FUNCTION_BLOCK FB_Mode
VAR_INPUT
	iManualMode:				BOOL; //manual button
	iAutoMode:					BOOL; //auto button
	iStartAutoCycle:			BOOL; //start auto cycle button
	iStopAutoCycle:				BOOL; //stop Auto cycle
	iStopEOC:					BOOL; //stop end of cycle
	iSemiAutoMode:				BOOL; //semi auto button
	iContCycle:					BOOL; //continuous cycle mode
	iSingleCycle:				BOOL; //single cycle mode
	iHome:						BOOL;  //station is at HOME
	iFault:						BOOL;
	iDryCycleMode:				BOOL; //station in dry cycle mode

	iIsStationSelected: BOOL; //is the current station selected?
	
	iLocalRemoteEnable: BOOL; //TRUE if the local station is in remote mode

	iRemoteData:typeRemote; //data from remote source
	
	iStartAutoCycleDelay:TIME:=T#2S; //delay time to start auto cycle
	iFirstScan:BOOL:=TRUE; //first scan logic for seting inital mode
	iStopCycleTimeout:TIME:=T#120S; //time to stop auto cycle if home not reached in (t). Set to 110% of expected station cycle time
	//isStationLocked:				BOOL;
END_VAR
	
	
VAR
	tAutoCycleStop: BOOL;
	timDelayRemoteOn: ton;
	ModeColourConv: FB_ModeStateToColour;
	timDelayAutoCycleStart: TON;
	timSEOCtimeout: TON;
	tUseOtherStation: BOOL;
	tResetSEOC: BOOL;
END_VAR

VAR_OUTPUT
END_VAR

VAR_IN_OUT
	stationState:typeStationMode;
	lockedModes:typeStationLockModes;
END_VAR
//theme:LYwABmhF6lY
VAR // added by the converter: edge detectors and wires of the graphical bodies
    _rt1, _rt2, _rt3, _rt4, _rt5, _rt6, _rt7, _rt8, _rt9, _rt10, _rt11, _rt12, _rt13, _rt14, _rt15, _rt16, _rt17, _rt18 : R_TRIG;
    _w1, _w2, _w3 : BOOL;
END_VAR

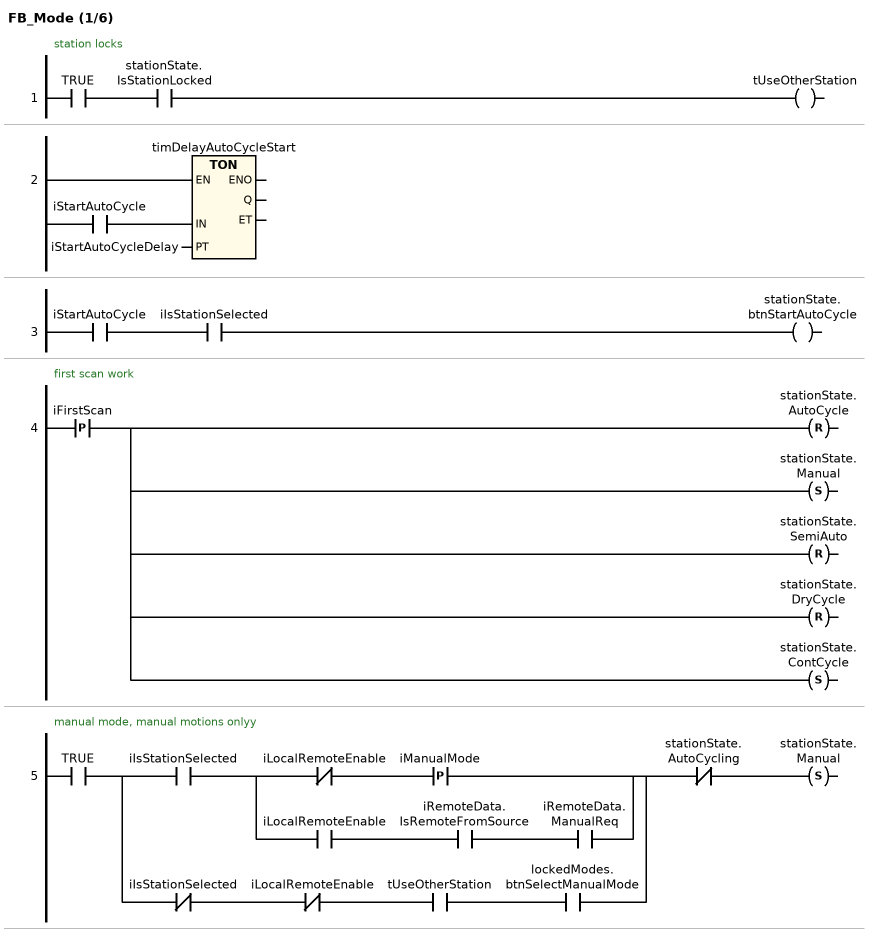
// NETWORK 1
// station locks
tUseOtherStation := TRUE AND stationState.IsStationLocked;

// NETWORK 2
timDelayAutoCycleStart(IN := iStartAutoCycle, PT := iStartAutoCycleDelay); // TON

// NETWORK 3
stationState.btnStartAutoCycle := iStartAutoCycle AND iIsStationSelected;

// NETWORK 4
// first scan work
_rt1(CLK := iFirstScan);
stationState.AutoCycle R= _rt1.Q;
stationState.Manual S= _rt1.Q;
stationState.SemiAuto R= _rt1.Q;
stationState.DryCycle R= _rt1.Q;
stationState.ContCycle S= _rt1.Q;

// NETWORK 5
// manual mode, manual motions onlyy
_rt2(CLK := iManualMode);
stationState.Manual S= TRUE AND (iIsStationSelected AND (NOT iLocalRemoteEnable AND _rt2.Q OR iLocalRemoteEnable AND iRemoteData.IsRemoteFromSource AND iRemoteData.ManualReq) OR NOT iIsStationSelected AND NOT iLocalRemoteEnable AND tUseOtherStation AND lockedModes.btnSelectManualMode) AND NOT stationState.AutoCycling;

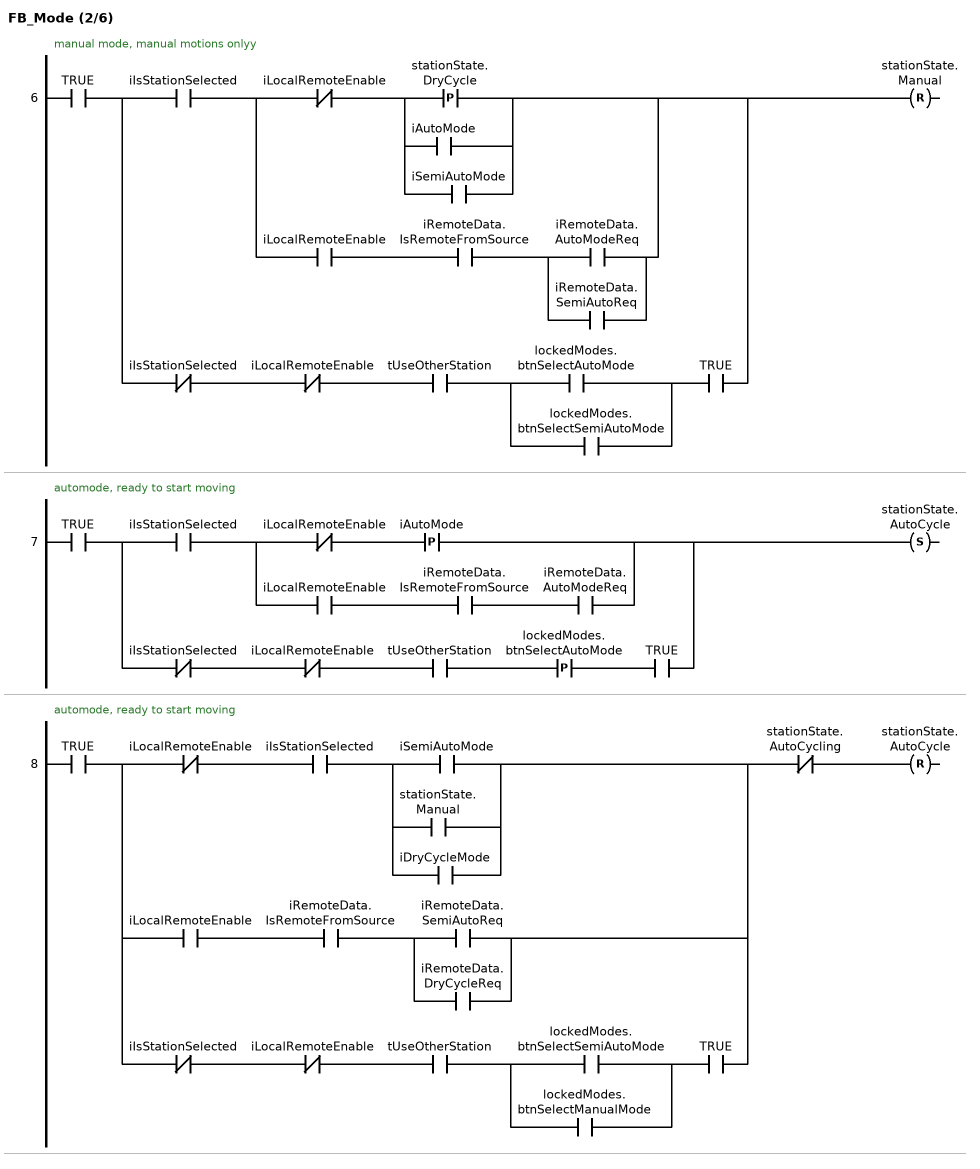
// NETWORK 6
// manual mode, manual motions onlyy
_rt3(CLK := stationState.DryCycle);
stationState.Manual R= TRUE AND (iIsStationSelected AND (NOT iLocalRemoteEnable AND (_rt3.Q OR iAutoMode OR iSemiAutoMode) OR iLocalRemoteEnable AND iRemoteData.IsRemoteFromSource AND (iRemoteData.AutoModeReq OR iRemoteData.SemiAutoReq)) OR NOT iIsStationSelected AND NOT iLocalRemoteEnable AND tUseOtherStation AND (lockedModes.btnSelectAutoMode OR lockedModes.btnSelectSemiAutoMode) AND TRUE);

// NETWORK 7
// automode, ready to start moving
_rt4(CLK := iAutoMode);
_rt5(CLK := lockedModes.btnSelectAutoMode);
stationState.AutoCycle S= TRUE AND (iIsStationSelected AND (NOT iLocalRemoteEnable AND _rt4.Q OR iLocalRemoteEnable AND iRemoteData.IsRemoteFromSource AND iRemoteData.AutoModeReq) OR NOT iIsStationSelected AND NOT iLocalRemoteEnable AND tUseOtherStation AND _rt5.Q AND TRUE);

// NETWORK 8
// automode, ready to start moving
stationState.AutoCycle R= TRUE AND (NOT iLocalRemoteEnable AND iIsStationSelected AND (iSemiAutoMode OR stationState.Manual OR iDryCycleMode) OR iLocalRemoteEnable AND iRemoteData.IsRemoteFromSource AND (iRemoteData.SemiAutoReq OR iRemoteData.DryCycleReq) OR NOT iIsStationSelected AND NOT iLocalRemoteEnable AND tUseOtherStation AND (lockedModes.btnSelectSemiAutoMode OR lockedModes.btnSelectManualMode) AND TRUE) AND NOT stationState.AutoCycling;

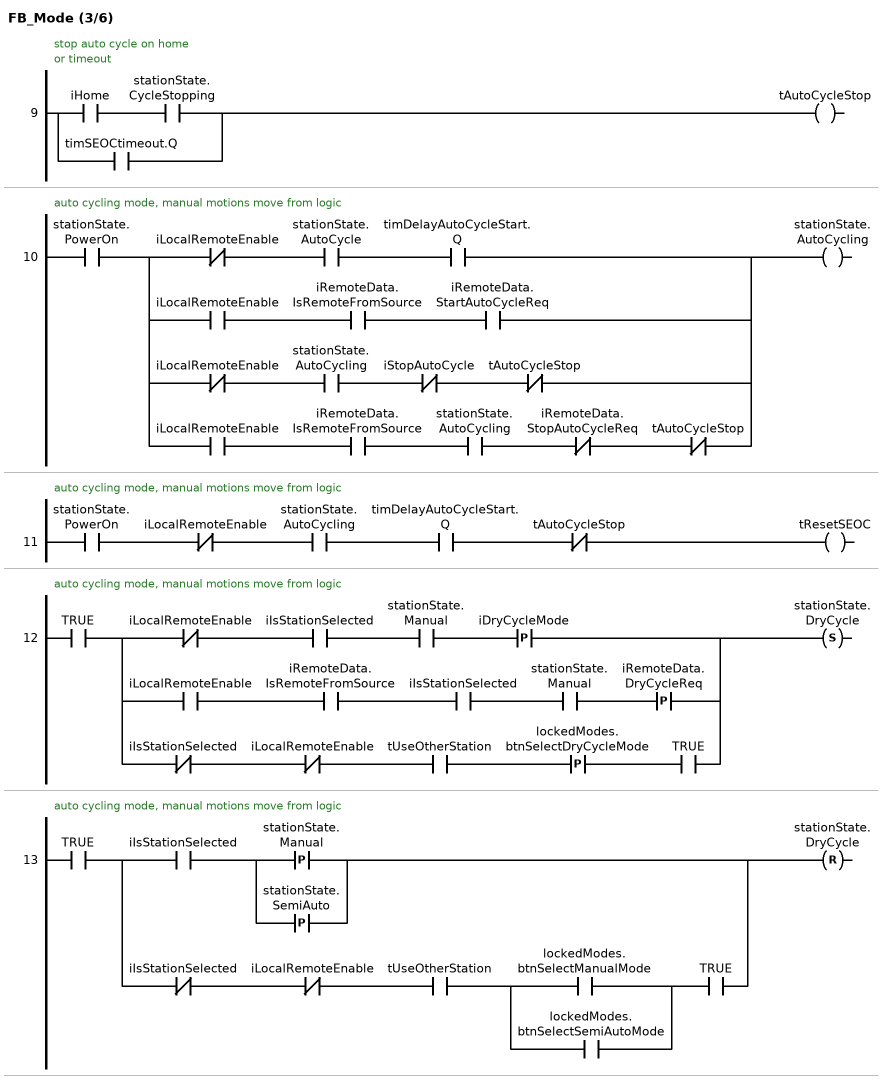
// NETWORK 9
// stop auto cycle on home
// or timeout
tAutoCycleStop := iHome AND stationState.CycleStopping OR timSEOCtimeout.Q;

// NETWORK 10
// auto cycling mode, manual motions move from logic
stationState.AutoCycling := stationState.PowerOn AND (NOT iLocalRemoteEnable AND stationState.AutoCycle AND timDelayAutoCycleStart.Q OR iLocalRemoteEnable AND iRemoteData.IsRemoteFromSource AND iRemoteData.StartAutoCycleReq OR NOT iLocalRemoteEnable AND stationState.AutoCycling AND NOT iStopAutoCycle AND NOT tAutoCycleStop OR iLocalRemoteEnable AND iRemoteData.IsRemoteFromSource AND stationState.AutoCycling AND NOT iRemoteData.StopAutoCycleReq AND NOT tAutoCycleStop);

// NETWORK 11
// auto cycling mode, manual motions move from logic
tResetSEOC := stationState.PowerOn AND NOT iLocalRemoteEnable AND stationState.AutoCycling AND timDelayAutoCycleStart.Q AND NOT tAutoCycleStop;

// NETWORK 12
// auto cycling mode, manual motions move from logic
_rt6(CLK := iDryCycleMode);
_rt7(CLK := iRemoteData.DryCycleReq);
_rt8(CLK := lockedModes.btnSelectDryCycleMode);
stationState.DryCycle S= TRUE AND (NOT iLocalRemoteEnable AND iIsStationSelected AND stationState.Manual AND _rt6.Q OR iLocalRemoteEnable AND iRemoteData.IsRemoteFromSource AND iIsStationSelected AND stationState.Manual AND _rt7.Q OR NOT iIsStationSelected AND NOT iLocalRemoteEnable AND tUseOtherStation AND _rt8.Q AND TRUE);

// NETWORK 13
// auto cycling mode, manual motions move from logic
_rt9(CLK := stationState.Manual);
_rt10(CLK := stationState.SemiAuto);
stationState.DryCycle R= TRUE AND (iIsStationSelected AND (_rt9.Q OR _rt10.Q) OR NOT iIsStationSelected AND NOT iLocalRemoteEnable AND tUseOtherStation AND (lockedModes.btnSelectManualMode OR lockedModes.btnSelectSemiAutoMode) AND TRUE);

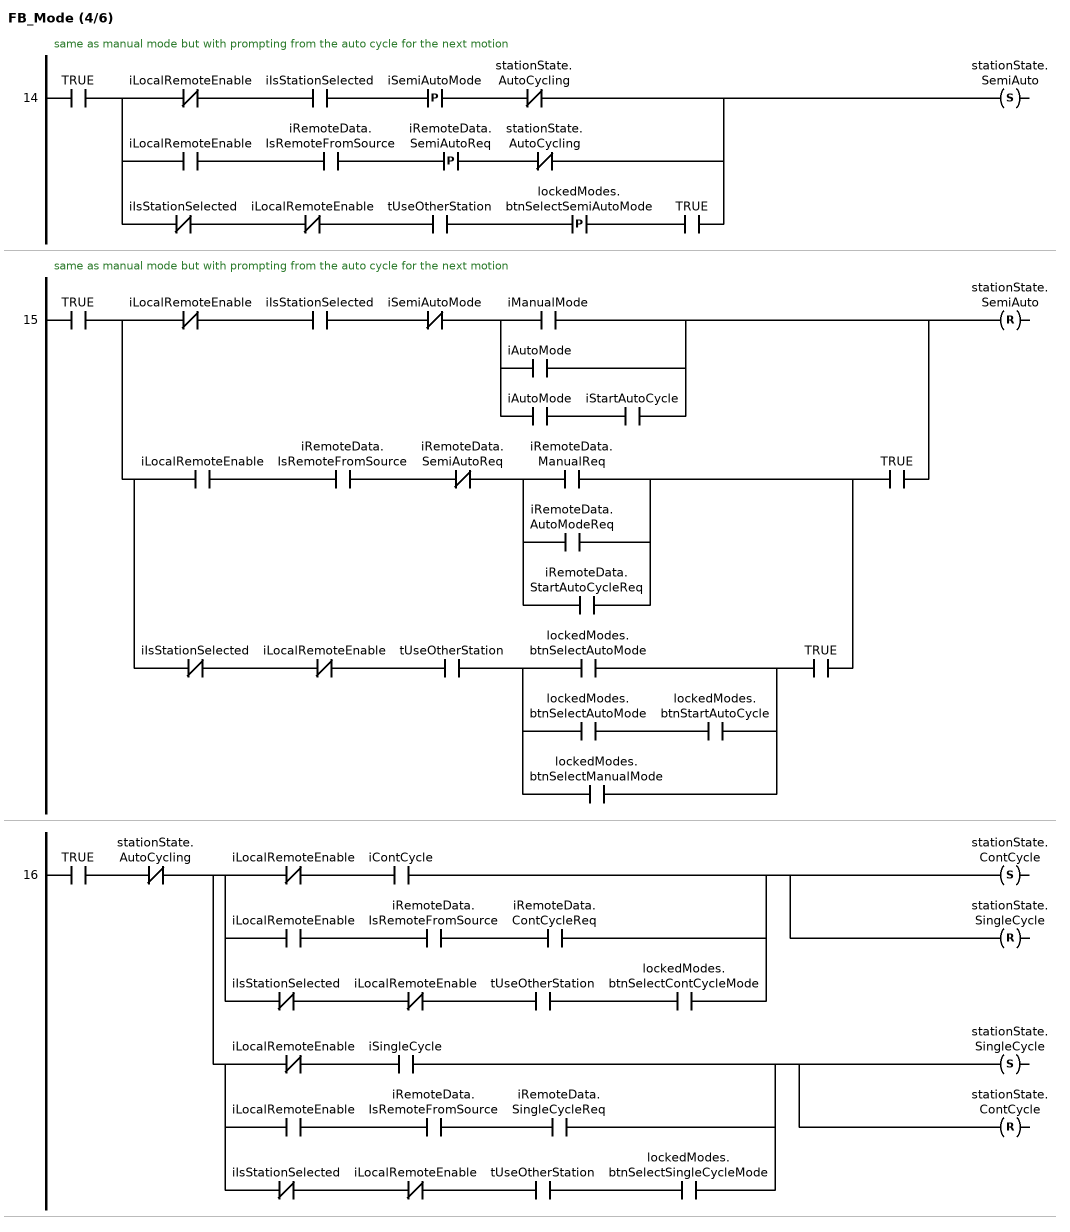
// NETWORK 14
// same as manual mode but with prompting from the auto cycle for the next motion
_rt11(CLK := iSemiAutoMode);
_rt12(CLK := iRemoteData.SemiAutoReq);
_rt13(CLK := lockedModes.btnSelectSemiAutoMode);
stationState.SemiAuto S= TRUE AND (NOT iLocalRemoteEnable AND iIsStationSelected AND _rt11.Q AND NOT stationState.AutoCycling OR iLocalRemoteEnable AND iRemoteData.IsRemoteFromSource AND _rt12.Q AND NOT stationState.AutoCycling OR NOT iIsStationSelected AND NOT iLocalRemoteEnable AND tUseOtherStation AND _rt13.Q AND TRUE);

// NETWORK 15
// same as manual mode but with prompting from the auto cycle for the next motion
stationState.SemiAuto R= TRUE AND (NOT iLocalRemoteEnable AND iIsStationSelected AND NOT iSemiAutoMode AND (iManualMode OR iAutoMode OR iAutoMode AND iStartAutoCycle) OR (iLocalRemoteEnable AND iRemoteData.IsRemoteFromSource AND NOT iRemoteData.SemiAutoReq AND (iRemoteData.ManualReq OR iRemoteData.AutoModeReq OR iRemoteData.StartAutoCycleReq) OR NOT iIsStationSelected AND NOT iLocalRemoteEnable AND tUseOtherStation AND (lockedModes.btnSelectAutoMode OR lockedModes.btnSelectAutoMode AND lockedModes.btnStartAutoCycle OR lockedModes.btnSelectManualMode) AND TRUE) AND TRUE);

// NETWORK 16
_w1 := TRUE AND NOT stationState.AutoCycling;
_w2 := _w1 AND (NOT iLocalRemoteEnable AND iContCycle OR iLocalRemoteEnable AND iRemoteData.IsRemoteFromSource AND iRemoteData.ContCycleReq OR NOT iIsStationSelected AND NOT iLocalRemoteEnable AND tUseOtherStation AND lockedModes.btnSelectContCycleMode);
stationState.ContCycle S= _w2;
stationState.SingleCycle R= _w2;
_w3 := _w1 AND (NOT iLocalRemoteEnable AND iSingleCycle OR iLocalRemoteEnable AND iRemoteData.IsRemoteFromSource AND iRemoteData.SingleCycleReq OR NOT iIsStationSelected AND NOT iLocalRemoteEnable AND tUseOtherStation AND lockedModes.btnSelectSingleCycleMode);
stationState.SingleCycle S= _w3;
stationState.ContCycle R= _w3;

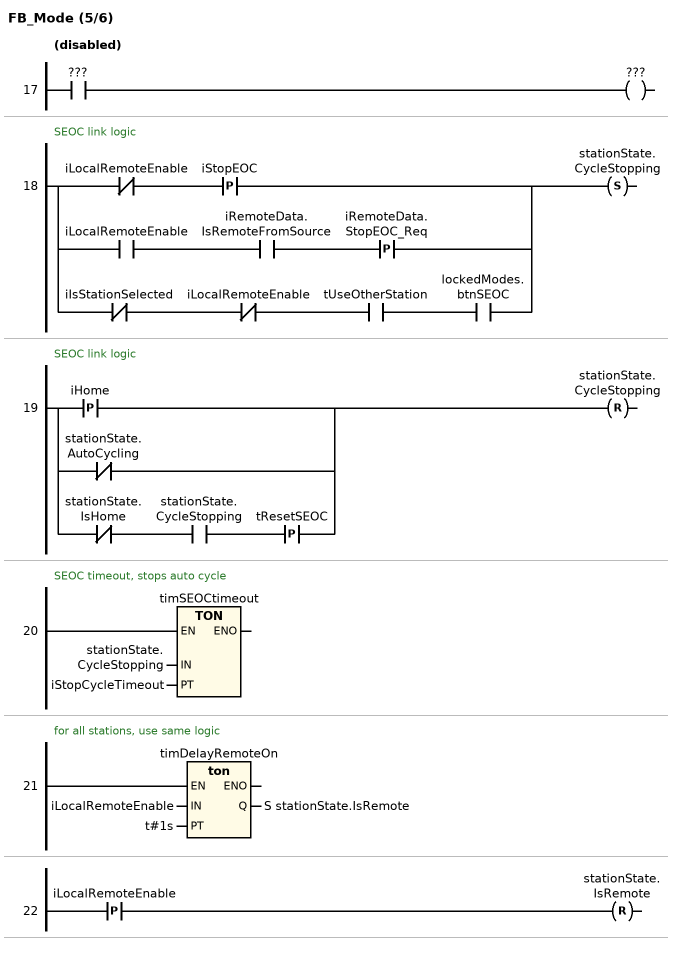
// NETWORK 17 (disabled)
// ??? := ???;

// NETWORK 18
// SEOC link logic
_rt14(CLK := iStopEOC);
_rt15(CLK := iRemoteData.StopEOC_Req);
stationState.CycleStopping S= NOT iLocalRemoteEnable AND _rt14.Q OR iLocalRemoteEnable AND iRemoteData.IsRemoteFromSource AND _rt15.Q OR NOT iIsStationSelected AND NOT iLocalRemoteEnable AND tUseOtherStation AND lockedModes.btnSEOC;

// NETWORK 19
// SEOC link logic
_rt16(CLK := iHome);
_rt17(CLK := tResetSEOC);
stationState.CycleStopping R= _rt16.Q OR NOT stationState.AutoCycling OR NOT stationState.IsHome AND stationState.CycleStopping AND _rt17.Q;

// NETWORK 20
// SEOC timeout, stops auto cycle
timSEOCtimeout(IN := stationState.CycleStopping, PT := iStopCycleTimeout); // TON

// NETWORK 21
// for all stations, use same logic
timDelayRemoteOn(IN := iLocalRemoteEnable, PT := t#1s); // ton
stationState.IsRemote S= timDelayRemoteOn.Q;

// NETWORK 22
_rt18(CLK := iLocalRemoteEnable);
stationState.IsRemote R= _rt18.Q;

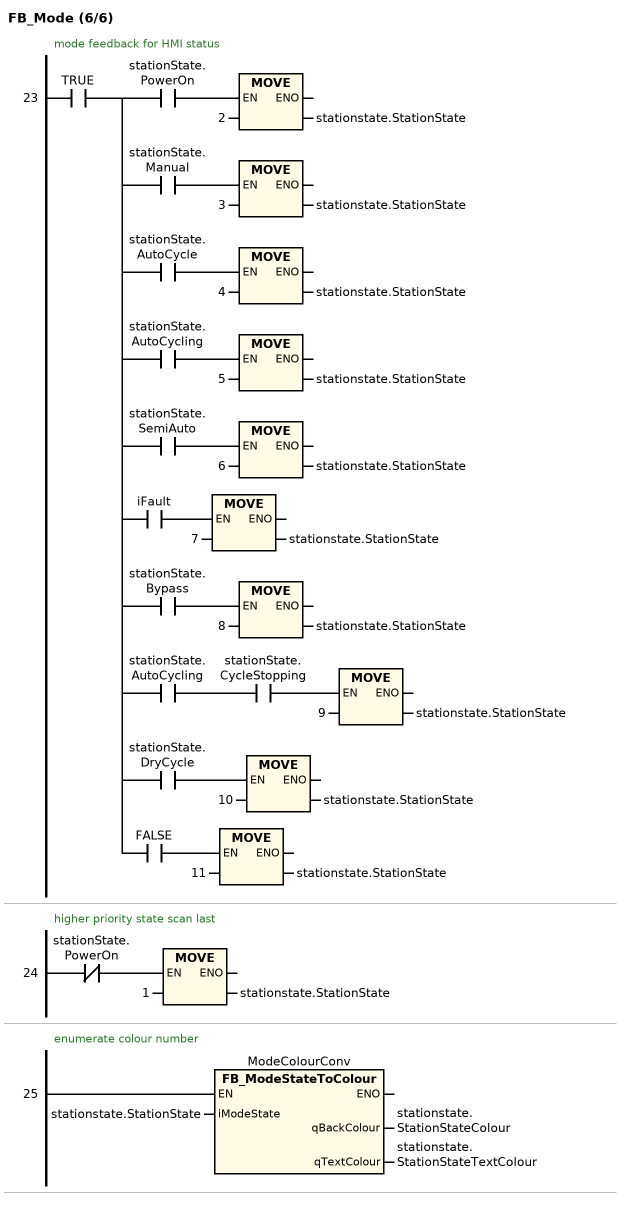
// NETWORK 23
// mode feedback for HMI status
IF TRUE AND stationState.PowerOn THEN stationstate.StationState := 2; END_IF
IF TRUE AND stationState.Manual THEN stationstate.StationState := 3; END_IF
IF TRUE AND stationState.AutoCycle THEN stationstate.StationState := 4; END_IF
IF TRUE AND stationState.AutoCycling THEN stationstate.StationState := 5; END_IF
IF TRUE AND stationState.SemiAuto THEN stationstate.StationState := 6; END_IF
IF TRUE AND iFault THEN stationstate.StationState := 7; END_IF
IF TRUE AND stationState.Bypass THEN stationstate.StationState := 8; END_IF
IF TRUE AND stationState.AutoCycling AND stationState.CycleStopping THEN stationstate.StationState := 9; END_IF
IF TRUE AND stationState.DryCycle THEN stationstate.StationState := 10; END_IF
IF TRUE AND FALSE THEN stationstate.StationState := 11; END_IF

// NETWORK 24
// higher priority state scan last
IF NOT stationState.PowerOn THEN stationstate.StationState := 1; END_IF

// NETWORK 25
// enumerate colour number
ModeColourConv(
    iModeState := stationstate.StationState,
    qBackColour => stationstate.StationStateColour,
    qTextColour => stationstate.StationStateTextColour); // FB_ModeStateToColour

END_FUNCTION_BLOCK

(* stored: Version 1.1.0.1, ProductVersion 3.1.4024.11
   POU FB_Mode: Id {ce08c7f1-a47e-41ce-a12a-5019455503c9}, SpecialFunc None *)
